FUNCTION_BLOCK FB_InnerCapillaryTubeMats EXTENDS FB_SystemContinous
VAR_INPUT
	bHeatingModeAutomatic : BOOL; //control mode: 0 = heating mode, 1 = cooling mode
	stAmbientState : ST_AmbientState;
END_VAR
VAR_OUTPUT
END_VAR
VAR
	{attribute 'OPC.UA.DA' := '1'}
	localSetParameters : ST_InnerCapillaryTubeMatsSetParameters;

	//default parameters
	localDefaultParameters : ST_InnerCapillaryTubeMatsDefaultParameters;	
	
	//pumps
	stPU405DefaultParameters : ST_PumpGrundfosMagna3DefaultParameters;
	stPU500DefaultParameters : ST_PumpGrundfosMagna3DefaultParameters;
	
	PU405 : FB_PumpGrundfosMagna3 := (ST_DefaultParameters := stPU405DefaultParameters);
	PU500 : FB_PumpGrundfosMagna3 := (ST_DefaultParameters := stPU500DefaultParameters);	
	
	//valves
	stSV401DefaultParameters : ST_DiscreteValveDefaultParameters := (nFeedback := 3);
	stSV402DefaultParameters : ST_DiscreteValveDefaultParameters := (nFeedback := 3);
	stSV403DefaultParameters : ST_DiscreteValveDefaultParameters := (nFeedback := 3);
	stSV404DefaultParameters : ST_DiscreteValveDefaultParameters := (nFeedback := 3);
	stRV500DefaultParameters : ST_MixingValveDefaultParameters := (bFeedbackSignal := FALSE, tTaskCycleTime := GlobalVariables.tCtrlCycleTime_MAIN, tCtrlCycleTime := GlobalVariables.tCtrlCycleTime_MAIN);	
	
	SV401 : FB_DiscreteValve := (ST_DefaultParameters := stSV401DefaultParameters); //cooling network supply
	SV402 : FB_DiscreteValve := (ST_DefaultParameters := stSV402DefaultParameters); //cooling network return
	SV403 : FB_DiscreteValve := (ST_DefaultParameters := stSV403DefaultParameters); //heating network supply
	SV404 : FB_DiscreteValve := (ST_DefaultParameters := stSV404DefaultParameters); //heating entwork return
	RV500 : FB_MixingValve := (ST_DefaultParameters := stRV500DefaultParameters);
	
	//internal variables
	bHeatingMode 			: BOOL;
	fOffSetTemperature		: REAL;
	bSetStatusOn_PU405 		: BOOL;
	bSetStatusOn_PU500 		: BOOL;
	bSetStatusOn_SV_CN 		: BOOL;
	bSetStatusOn_SV_HNLT	: BOOL;
	bSetStatusOn_RV500 		: BOOL;
	fSetPoint_RV500 		: REAL;
	nControlMode_RV500 		: E_MixingValveControlMode;
	
	//characteristic curves
	CharacteristicCurve 			: FB_CTRL_FLOW_TEMP_SETPOINT_GEN;
	CharacteristicCurve_Parameters	: ST_CTRL_FLOW_TEMP_SETPOINT_GEN_PARAMS;
	
	//triggers
	SwitchToHeating : R_TRIG;
	SwitchToCooling : F_TRIG;
	bFinishedSwitchMode : BOOL := TRUE;
	
	//clock
	stDefaultParameters_Clock : ST_ClockDefaultParameters := (tTaskCycleTime := GlobalVariables.tCtrlCycleTime_MAIN, tCtrlCycleTime := T#1M);
	Clock : FB_Clock := (ST_DefaultParameters := stDefaultParameters_Clock);
END_VAR

//check if heating mode has switched
SelectInnerCapillaryTubeMatsControlMode();
SwitchToHeating(CLK := bHeatingMode);
SwitchToCooling(CLK := bHeatingMode);

//MAIN must be called before SwitchMode to prevent pump signal chattering (signal is written after SwitchMode function)
MAIN();

//disrupt calling SystemFlowControl via MAIN() when mode is switched and call SwitchMode()
IF (SwitchToHeating.Q OR SwitchToCooling.Q) OR NOT bFinishedSwitchMode THEN
	SwitchMode(bSwitchToHeating := SwitchToHeating.Q AND NOT SwitchToCooling.Q,
		bFinishedSwitchMode => bFinishedSwitchMode);
END_IF;


//clock for night setback
Clock();

//pumps
PU405.GetState_Profibus();
PU405(bSetStatusOnAutomatic := bSetStatusOn_PU405,
	fSetPointAutomatic := 70,
	bAlgorithmPermission := bAlgorithmPermission,
	nControlModeAutomatic := 0);
PU405.SetState_Profibus();

PU500.GetState_Profibus();
PU500(bSetStatusOnAutomatic := bSetStatusOn_PU500,
	fSetPointAutomatic := 70,
	bAlgorithmPermission := bAlgorithmPermission,
	nControlModeAutomatic := 0);
PU500.SetState_Profibus();

//valves
SV401.GetState_BI();
SV401(bSetStatusOnAutomatic := bSetStatusOn_CN,
	bAlgorithmPermission := bAlgorithmPermission);
SV401.SetState_BO();

SV402.GetState_BI();
SV402(bSetStatusOnAutomatic := bSetStatusOn_CN,
	bAlgorithmPermission := bAlgorithmPermission);
SV402.SetState_BO();

SV403.GetState_BI();
SV403(bSetStatusOnAutomatic := bSetStatusOn_HNLT,
	bAlgorithmPermission := bAlgorithmPermission);
SV403.SetState_BO();

SV404.GetState_BI();
SV404(bSetStatusOnAutomatic := bSetStatusOn_HNLT,
	bAlgorithmPermission := bAlgorithmPermission);
SV404.SetState_BO();

RV500.GetState_AI();
RV500(bSetStatusOnAutomatic := bSetStatusOn_RV500,
	fSetPointAutomatic := fSetPoint_RV500,
	bAlgorithmPermission := bAlgorithmPermission,
	fTemperatureExternal := PU500.fTemperatureExternal,
	nControlModeAutomatic := nControlMode_RV500);
RV500.SetState_AO();

METHOD PRIVATE ControlInnerCapillaryTubeMats : BOOL
VAR_INPUT
END_VAR
VAR
END_VAR
CharacteristicCurve_Parameters.fAmbientTempMax := localDefaultParameters.aLimitsAmbientTemperature[2];
CharacteristicCurve_Parameters.fAmbientTempMin := localDefaultParameters.aLimitsAmbientTemperature[1];
CharacteristicCurve_Parameters.fForeRunTempMax := localDefaultParameters.aLimitsFeedTemperature[1];
CharacteristicCurve_Parameters.fForeRunTempMin := localDefaultParameters.aLimitsFeedTemperature[2];
CharacteristicCurve_Parameters.tCtrlCycleTime := GlobalVariables.tCtrlCycleTime_MAIN;
CharacteristicCurve_Parameters.tTaskCycleTime := GlobalVariables.tTaskCycleTime_MAIN;

//calculate offset temperature depending on heating or cooling mode and daytime
IF Clock.stClockState.fHour>19 AND Clock.stClockState.fHour<7 THEN
	IF bHeatingMode THEN
		fOffSetTemperature := -localDefaultParameters.fNightSetback;
	ELSE
		fOffSetTemperature := localDefaultParameters.fNightSetback;
	END_IF
ELSE
	fOffSetTemperature := 0;
END_IF

CharacteristicCurve(fAmbientTemperature := stAmbientState.fOutsideTemperature,
	fOffsetTemperature := fOffSetTemperature,
	bLimitFlowTemp := TRUE,
	stParams := CharacteristicCurve_Parameters);
fSetPoint_RV500 := CharacteristicCurve.fOut;
END_METHOD

METHOD PROTECTED  Operational : BOOL
VAR_INPUT
END_VAR
VAR_OUTPUT
	bSwitchToWorking : BOOL := FALSE;
END_VAR
END_METHOD

METHOD PROTECTED  RampDown : BOOL
VAR_INPUT
END_VAR
VAR_OUTPUT
	bRampDownFinished : BOOL := FALSE;
END_VAR
END_METHOD

METHOD PROTECTED  RampUp : BOOL
VAR_INPUT
END_VAR
VAR_OUTPUT
	bRampUpFinished : BOOL := FALSE;
END_VAR
END_METHOD

METHOD PRIVATE SelectInnerCapillaryTubeMatsControlMode : BOOL
VAR_INPUT
END_VAR
IF control.bManualModeActivated THEN
	bHeatingMode := localSetParameters.bHeatingModeManual;
ELSIF control.bAlgorithmModeActivated AND bAlgorithmPermission THEN
	bHeatingMode := localSetParameters.bHeatingModeAlgorithm;
ELSE
	bHeatingMode := bHeatingModeAutomatic;
END_IF
END_METHOD

METHOD PRIVATE SwitchMode : BOOL
VAR_INPUT
	bSwitchToHeating : BOOL; //if false switch to cooling
END_VAR
VAR_OUTPUT
	bFinishedSwitchMode : BOOL := FALSE;
END_VAR
VAR_INST
	bRampDownFinished : BOOL := FALSE;
END_VAR
//check system state
IF bRampDownFinished THEN
	IF bSwitchToHeating THEN
		//close valve in cooling network
		bSetStatusOn_SV_CN := FALSE;
		//wait until valves in cooling network are closed before opening valves in heating network
		IF NOT SV401.bStatusOn AND NOT SV402.bStatusOn THEN
			bSetStatusOn_SV_HNLT := TRUE;		
		END_IF
		IF SV403.bStatusOn AND SV404.bStatusOn THEN
			//reset instant variable
			bRampDownFinished := FALSE;			
			bFinishedSwitchMode := TRUE;
		END_IF
		
	ELSE
		//close valve in heating network
		bSetStatusOn_SV_HNLT := FALSE;
		//wait until valves in heating network are closed before opening valves in cooling network
		IF NOT SV403.bStatusOn AND NOT SV404.bStatusOn THEN
			bSetStatusOn_SV_CN := TRUE;		
		END_IF
		IF SV401.bStatusOn AND SV402.bStatusOn THEN
			bFinishedSwitchMode := TRUE;
			//reset instant variable
			bRampDownFinished := FALSE;
		END_IF
	END_IF
ELSE
	RampDown(bRampDownFinished => bRampDownFinished);
END_IF
END_METHOD

METHOD PROTECTED  Working : BOOL
VAR_INPUT
END_VAR
VAR_OUTPUT
	bSwitchToOperational : BOOL := FALSE;
END_VAR
END_METHOD

END_FUNCTION_BLOCK

(* stored: Version 1.1.0.1, ProductVersion 3.1.4024.10
   POU FB_InnerCapillaryTubeMats: Id {46ec983e-b705-43aa-aa03-31694ea1c351}, SpecialFunc None
   Method ControlInnerCapillaryTubeMats: Id {4d780eb0-c994-49a4-a3af-4cc20bccd6d0}
   Method Operational: Id {e9dd841f-7be7-4729-ab2a-e0444d4793cf}
   Method RampDown: Id {a3bbb3df-240d-4274-b5c7-44e29ede78a1}
   Method RampUp: Id {9c85ac6b-2d18-4fd9-84e6-e871c2d86ae0}
   Method SelectInnerCapillaryTubeMatsControlMode: Id {c6246abd-6c96-45f1-8bcd-105c886c486e}
   Method SwitchMode: Id {454a6e9c-2859-4a72-a2fb-db3e1e6f3e67}
   Method Working: Id {a6a11e5f-819e-494c-8b28-af1733451e25} *)
